// TIA Portal project "2022.11.03—成绩录入、重置" (V17)

(* hardware
DEVICE "S7-1200 station_1"  S7-1200 Station
   slot 0: "Rack_0"  S7-1200 Rack  Rack  V1.0
   slot 1: "PLC_1"  CPU 1214C DC/DC/Rly  6ES7 214-1HG40-0XB0  V4.5
DEVICE "HMI_1"  KTP700 Basic PN
   slot 0: "HMI_1"  KTP700 Basic PN  6AV2 123-2GB03-0AX0  17.0.0.0
   slot 1: "HMI_RT_1"  KTP700 Basic PN  6AV2 123-2GB03-0AX0  17.0.0.0
   slot 5: "HMI_1.IE_CP_1"  PROFINET Interface  17.0.0.0
      slot 1: "PROFINET Interface_1"  PROFINET Interface
         slot 1: "Port_1"  Port
*)

// ===== PLC "PLC_1"  CPU 1214C DC/DC/Rly =====

DATA_BLOCK "数据块_1"   // DB1
{ S7_Optimized_Access := 'TRUE' }
VERSION : 0.1
   VAR
      day_time : DTL;
      RETURN_VAL : Int;
      中间变量1 : DInt;
      中间变量2 : Real;
      中间变量3 : Real;
      中间变量4 : UDInt;
      中间变量5 : Real;
      中间变量6 : DInt;
      中间变量7 : UDInt;
      "Randow-score" : UDInt;
      待录入成绩 : UDInt;
      总成绩 : UDInt;
      平均值 : Real;
      取平均值 : Bool;
      随机生成成绩 : Bool;
      手动录入成绩 : Bool;
      初始化 : Bool;
      操作数1 : Bool;
      操作数2 : Bool;
      操作数3 : Bool;
      操作数4 : Bool;
      运行标记 : UDInt;
      Score : Array[1..10] of UDInt;
      "index 1" : DInt := 1;
      "index 2" : DInt := 1;
   END_VAR
BEGIN
END_DATA_BLOCK

ORGANIZATION_BLOCK "Main"   // OB1, LAD, ProgramCycle
TITLE = "Main Program Sweep (Cycle)"
{ S7_Optimized_Access := 'TRUE' }
VERSION : 0.1
   VAR_INPUT
      Initial_Call : Bool;   // Initial call of this OB
      Remanence : Bool;   // =True, if remanent data are available
   END_VAR
   VAR_TEMP   // added for the SCL form of the ladder/FBD networks
      _w1 : Bool;
      _w2 : Bool;
      _w3 : Bool;
      _w4 : Bool;
   END_VAR
BEGIN

REGION Network 1
   // 取纳秒前两个数或后两个数  用move取出 纳秒  conv转换类型      除数取前两位  取整
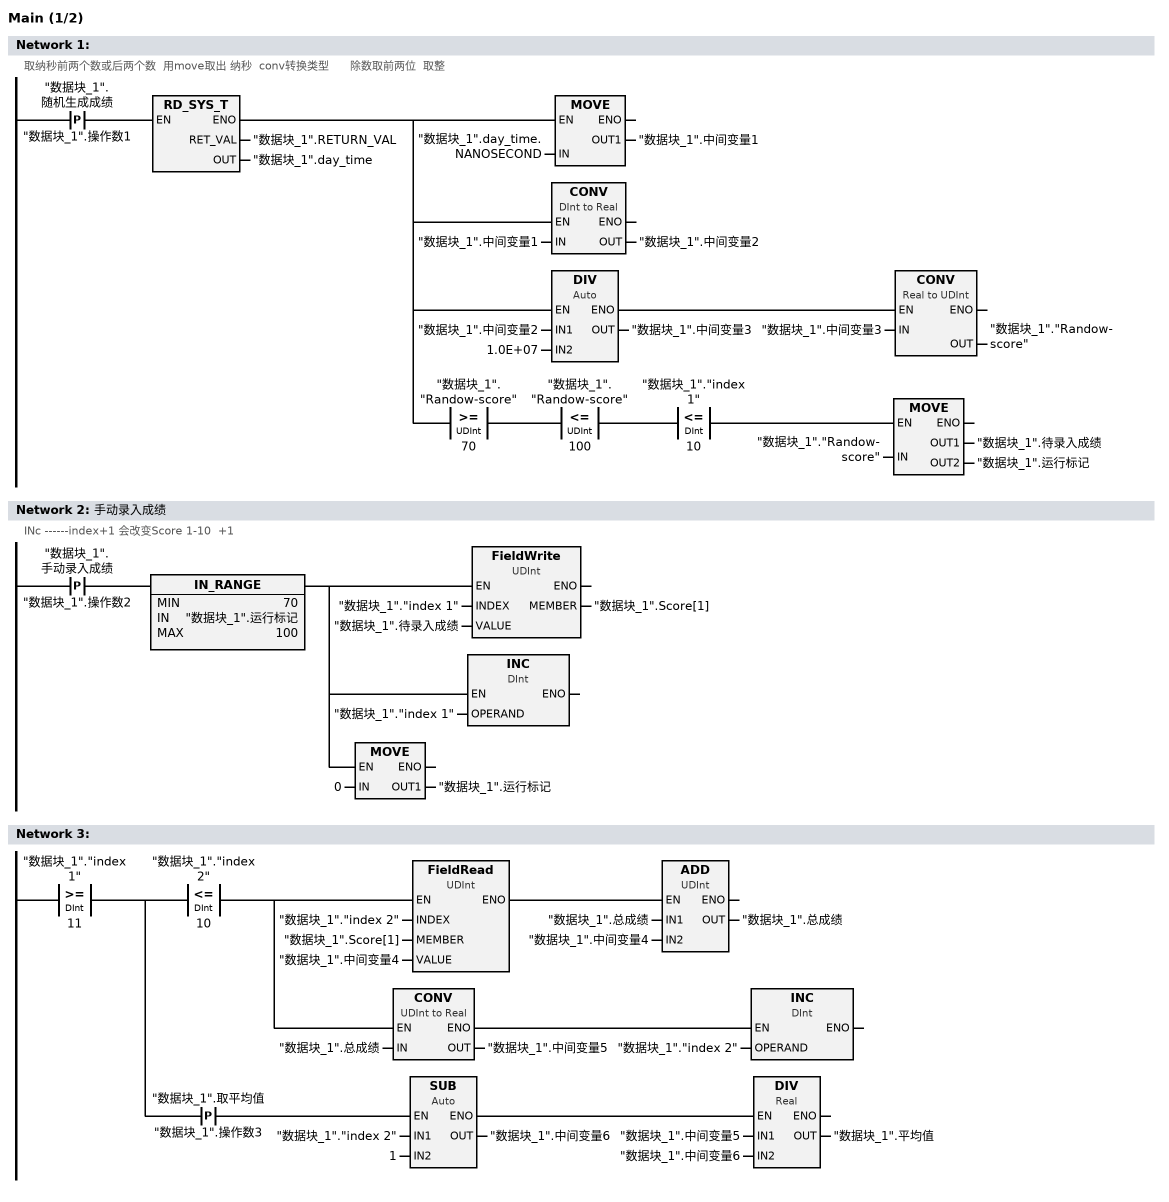
   // ENO of a box is taken as its EN; it also drops when the box reports an error
   #_w1 := "数据块_1".随机生成成绩 AND NOT "数据块_1".操作数1;   // rising edge of "数据块_1".随机生成成绩
   "数据块_1".操作数1 := "数据块_1".随机生成成绩;
   IF #_w1 THEN
       "数据块_1".RETURN_VAL := RD_SYS_T(OUT => "数据块_1".day_time);
       "数据块_1".中间变量1 := "数据块_1".day_time.NANOSECOND;
       "数据块_1".中间变量2 := DINT_TO_REAL("数据块_1".中间变量1);
       "数据块_1".中间变量3 := "数据块_1".中间变量2 / 1.0E+07;
       "数据块_1"."Randow-score" := REAL_TO_UDINT("数据块_1".中间变量3);
   END_IF;
   IF #_w1 AND ("数据块_1"."Randow-score" >= 70) AND ("数据块_1"."Randow-score" <= 100) AND ("数据块_1"."index 1" <= 10) THEN
       "数据块_1".待录入成绩 := "数据块_1"."Randow-score";
       "数据块_1".运行标记 := "数据块_1"."Randow-score";
   END_IF;
END_REGION

REGION Network 2: 手动录入成绩
   // INc ------index+1 会改变Score 1-10  +1
   // no SCL statement known for FieldWrite: written as a call
   #_w1 := "数据块_1".手动录入成绩 AND NOT "数据块_1".操作数2;   // rising edge of "数据块_1".手动录入成绩
   "数据块_1".操作数2 := "数据块_1".手动录入成绩;
   #_w2 := #_w1 AND (70 <= "数据块_1".运行标记) AND ("数据块_1".运行标记 <= 100);
   IF #_w2 THEN
       FieldWrite(index := "数据块_1"."index 1", value := "数据块_1".待录入成绩, member => "数据块_1".Score[1]);
       "数据块_1"."index 1" := "数据块_1"."index 1" + 1;
       "数据块_1".运行标记 := 0;
   END_IF;
END_REGION

REGION Network 3
   // no SCL statement known for FieldRead: written as a call
   // ENO of a box is taken as its EN; it also drops when the box reports an error
   #_w1 := "数据块_1"."index 1" >= 11;
   #_w2 := #_w1 AND ("数据块_1"."index 2" <= 10);
   #_w3 := #_w1 AND ("数据块_1"."index 2" <= 10);
   IF #_w3 THEN
       FieldRead(index := "数据块_1"."index 2", member := "数据块_1".Score[1], value := "数据块_1".中间变量4);
       "数据块_1".总成绩 := "数据块_1".总成绩 + "数据块_1".中间变量4;
   END_IF;
   IF #_w2 THEN
       "数据块_1".中间变量5 := UDINT_TO_REAL("数据块_1".总成绩);
       "数据块_1"."index 2" := "数据块_1"."index 2" + 1;
   END_IF;
   #_w4 := #_w1 AND "数据块_1".取平均值 AND NOT "数据块_1".操作数3;   // rising edge of "数据块_1".取平均值
   "数据块_1".操作数3 := "数据块_1".取平均值;
   IF #_w4 THEN
       "数据块_1".中间变量6 := "数据块_1"."index 2" - 1;
       "数据块_1".平均值 := "数据块_1".中间变量5 / "数据块_1".中间变量6;
   END_IF;
END_REGION

REGION Network 4: 初始化
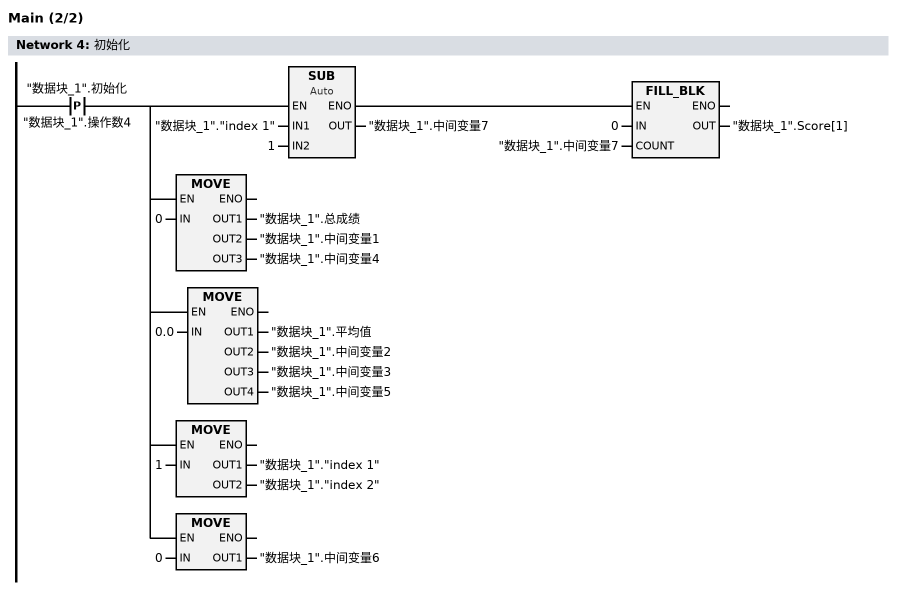
   RUNG wire#powerrail
      P_Contact(operand := "数据块_1".初始化, bit := "数据块_1".操作数4)
      wire#w1
      Sub(in1 := "数据块_1"."index 1", in2 := 1, out => "数据块_1".中间变量7)
      FillBlockI(in := 0, count := "数据块_1".中间变量7, out => "数据块_1".Score[1])
   END_RUNG
   RUNG wire#w1
      Move(in := 0, out1 => "数据块_1".总成绩, out2 => "数据块_1".中间变量1, out3 => "数据块_1".中间变量4)
   END_RUNG
   RUNG wire#w1
      Move(in := 0.0, out1 => "数据块_1".平均值, out2 => "数据块_1".中间变量2, out3 => "数据块_1".中间变量3, out4 => "数据块_1".中间变量5)
   END_RUNG
   RUNG wire#w1
      Move(in := 1, out1 => "数据块_1"."index 1", out2 => "数据块_1"."index 2")
   END_RUNG
   RUNG wire#w1
      Move(in := 0, out1 => "数据块_1".中间变量6)
   END_RUNG
   // the same network as SCL:
   #_w1 := "数据块_1".初始化 AND NOT "数据块_1".操作数4;   // rising edge of "数据块_1".初始化
   "数据块_1".操作数4 := "数据块_1".初始化;
   IF #_w1 THEN
       "数据块_1".中间变量7 := "数据块_1"."index 1" - 1;
       FILL_BLK(IN := 0, COUNT := "数据块_1".中间变量7, OUT => "数据块_1".Score[1]);
       "数据块_1".总成绩 := 0;
       "数据块_1".中间变量1 := 0;
       "数据块_1".中间变量4 := 0;
       "数据块_1".平均值 := 0.0;
       "数据块_1".中间变量2 := 0.0;
       "数据块_1".中间变量3 := 0.0;
       "数据块_1".中间变量5 := 0.0;
       "数据块_1"."index 1" := 1;
       "数据块_1"."index 2" := 1;
       "数据块_1".中间变量6 := 0;
   END_IF;
END_REGION
END_ORGANIZATION_BLOCK

(* ===== HMI "HMI_RT_1" =====
system functions are stored by id; their names below are inferred from use
connection "HMI_连接_1": ETHERNET, SMART_S7_1200_OMS

HMI tags "默认变量表"
   "Tag_ScreenNumber" : UInt, internal
   "数据块_1_随机生成成绩" : Bool = PLC 数据块_1.随机生成成绩, 1 s
   "数据块_1_手动录入成绩" : Bool = PLC 数据块_1.手动录入成绩, 1 s
   "数据块_1_取平均值" : Bool = PLC 数据块_1.取平均值, 1 s
   "数据块_1_初始化" : Bool = PLC 数据块_1.初始化, 1 s
   "数据块_1_待录入成绩" : UDInt = PLC 数据块_1.待录入成绩, 1 s
   "数据块_1_平均值" : Real = PLC 数据块_1.平均值, 1 s
   "数据块_1_index 1" : DInt = PLC 数据块_1."index 1", 1 s

Template "模板_1" 800x480
   Button "退出" at 714,429 size 71x50; TextOff '退出'; PictureOff "ExitRuntime_KTP700_Basic_PN_TR"; PictureOn "ExitRuntime_KTP700_Basic_PN_TR"
      on Release: StopRuntime(0)
   Button "Template_Button" at 614,429 size 71x50; TextOff 'Text'
   Button "Template_Button_1" at 514,429 size 71x50; TextOff 'Text'
   Button "Template_Button_2" at 414,429 size 71x50; TextOff 'Text'
   Button "Template_Button_3" at 314,429 size 71x50; TextOff 'Text'
   Button "Template_Button_4" at 214,429 size 71x50; TextOff 'Text'
   Button "报警" at 114,429 size 71x50; TextOff '报警'; PictureOff "AlarmDisplay_KTP700_Basic_PN_TR"; PictureOn "AlarmDisplay_KTP700_Basic_PN_TR"
      on Release: function_ef3f5d25("报警窗口_Unacknowledged", -1)
   Button "起始画面" at 14,429 size 71x50; TextOff '起始画面'; PictureOff "NavigateHome_KTP700_Basic_PN_TR"; PictureOn "NavigateHome_KTP700_Basic_PN_TR"
      on Release: ActivateScreen("根画面", 0)
   SymbolicIOField "Symbolic_IO_Field_Screen" at 93,9 size 600x33; TextOff '0'; TextOn '1'; TextList "TextList_ScreenNames"
      ProcessValue <- "Tag_ScreenNumber"
      on Change: ActivateScreenByNumber("Tag_ScreenNumber", 0)
   DateTimeField "HmiScreenItemData" at 695,25 size 105x25
   DateTimeField "HmiScreenItemData_1" at 695,0 size 105x25
   GraphicView "Logo" at 0,0 size 91x51; Picture "HMI_1 的 Logo"

screen "根画面" 800x480, template "模板_1"
   on GenerateScreen: SetTag("Tag_ScreenNumber", 1)
   Button "按钮_1" at 233,195 size 118x32; TextOff '随机生成成绩'
      on Press: SetBit("数据块_1_随机生成成绩")
      on Release: ResetBit("数据块_1_随机生成成绩")
   Button "按钮_2" at 235,248 size 117x32; TextOff '手动录入成绩'
      on Release: ResetBit("数据块_1_手动录入成绩")
      on Press: SetBit("数据块_1_手动录入成绩")
   Button "按钮_3" at 428,198 size 119x32; TextOff '获取平均成绩'
      on Press: SetBit("数据块_1_取平均值")
      on Release: ResetBit("数据块_1_取平均值")
   Button "按钮_4" at 427,247 size 119x32; TextOff '重置成绩'
      on Press: SetBit("数据块_1_初始化")
      on Release: ResetBit("数据块_1_初始化")
   IOField "I/O 域_1" at 220,128 size 145x32; FormatPattern 9999999999
      ProcessValue <- "数据块_1_待录入成绩"
   IOField "I/O 域_2" at 417,129 size 144x32; FormatPattern s999999999.999
      ProcessValue <- "数据块_1_平均值"
   TextField "文本域_1" at 245,96 size 90x20; Text '待录入成绩'
   TextField "文本域_2" at 453,101 size 73x20; Text '平均成绩'
   TextField "文本域_3" at 196,323 size 434x37; Text '成绩录入完成，获取平均成绩'
      Visibility <- "数据块_1_index 1"
*)